ABB RobotStudio station: SemesterProjekt_sim.rsstn

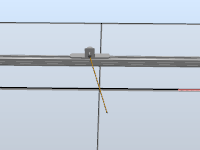
Station SemesterProjekt_sim (saved by RobotStudio 7.0.8728.594)
Layout (positions relative to the parent item):
  - BaseConstruktion [part] at (-0.03, 0.43, 41.45) mm, rotated rx 89.99 ry 0 rz -0.01 deg
  - Cart [part] at (1538.4, 109.33, 431.45) mm, rotated rx 89.99 ry 0 rz -0.01 deg
  - endBlock [part] at (0, -450, 0) mm, rotated rx 90 ry 0 rz 0 deg
  - Part_7 [part] at (2080, 325.44, 436.4) mm, rotated rx 0 ry 0 rz 90 deg
  - Part_8 [part] at (40, 325.44, 436.4) mm, rotated rx 0 ry 0 rz 90 deg
  - pendu [part] at (1938.39, 384.3, 466.37) mm, rotated rx -179.96 ry -0.17 rz -180 deg
